{attribute 'linkalways'} 
{attribute 'no_explicit_call' := 'This FB is a CLASS and must be accessed using methods or properties'}
{attribute 'enable_dynamic_creation'}
FUNCTION_BLOCK FINAL SEL_DINT EXTENDS Node
VAR
	g : _BOOL(FALSE);
	in1 : _DINT(0);
	in2 : _DINT(0);
	out : _DINT(0);
END_VAR

METHOD PUBLIC Clone : I_Node
VAR
	pNode : POINTER TO SEL_DINT;
END_VAR
pNode := __NEW(SEL_DINT);
Clone := pNode^;
END_METHOD

METHOD FB_init : BOOL
VAR_INPUT
	bInitRetains : BOOL; // if TRUE, the retain variables are initialized (warm start / cold start)
	bInCopyCode : BOOL;  // if TRUE, the instance afterwards gets moved into the copy code (online change)
END_VAR
AddInput('g',THIS^.g);
AddInput('in1',THIS^.in1);
AddInput('in2',THIS^.in2);
AddOutput('out', THIS^.out);
END_METHOD

METHOD PROTECTED OnExecute
VAR
END_VAR
IF g.value THEN
	out.value := in2.value;
ELSE
	out.value := in1.value;
END_IF
END_METHOD

END_FUNCTION_BLOCK

(* stored: Version 1.1.0.1, ProductVersion 3.1.4024.15
   POU SEL_DINT: Id {cd7f3716-c572-49dd-bba0-0b4e8efac401}, SpecialFunc None
   Folder Constructor: Id {1bb13929-fcfc-4009-bb59-386539dd0d99}
   Method Clone: Id {c9ce0f3e-1594-4549-95f8-7bafd7a3fe4b}
   Method FB_init: Id {e2314810-d1c3-4592-b36c-0358f738a59c}
   Method OnExecute: Id {959a1974-ae40-4650-9bab-191d31b01cb8} *)
